(* Logix 5000 project; controller test4 1769-L16ER-BB1B rev 36.11; software revision 36.00 *)

TASK MainTask (continuous, watchdog 500 ms) : MainProgram

MODULES
   Local : 1769-L16ER-BB1B (PointIO 0, rev 36.11)
      Discrete_IO : Embedded (PointIO 1, rev 36.11, Output RPI 20 ms)
           Local:1:I.Data.1   // Button 2
           Local:1:I.Data.2   // Button 3
           Local:1:I.Data.3   // Button 4
           Local:1:I.Data.4   // Switch 1
           Local:1:O.Data.0   // Light 1
           Local:1:O.Data.1   // Light 2
END_MODULES

PROGRAM MainProgram   (* main routine MainRoutine *)
VAR
   Green_Button : ALIAS FOR Local:1:I.Data.0;
   GreenButton : ALIAS FOR Local:1:I.Data.0;
   Timer1 : TIMER := (PRE := 4000, ACC := 1);
END_VAR

ROUTINE FBD1   (* function block diagram *)
   SHEET 1
END_ROUTINE

ROUTINE MainRoutine   (* ladder *)
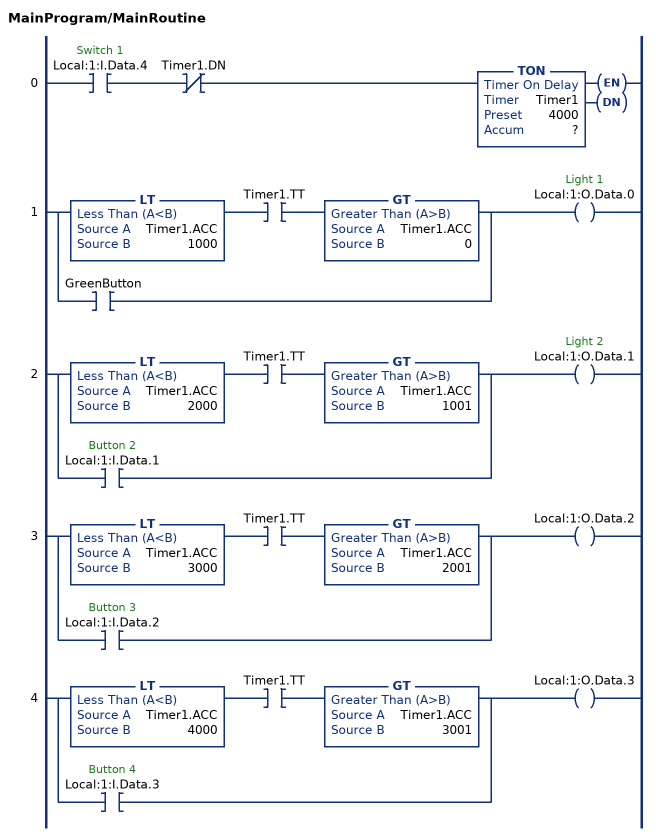
   0: XIC(Local:1:I.Data.4)XIO(Timer1.DN)TON(Timer1,?,?);
   1: [LT(Timer1.ACC,1000) XIC(Timer1.TT) GT(Timer1.ACC,0) ,XIC(GreenButton) ]OTE(Local:1:O.Data.0);
   2: [LT(Timer1.ACC,2000) XIC(Timer1.TT) GT(Timer1.ACC,1001) ,XIC(Local:1:I.Data.1) ]OTE(Local:1:O.Data.1);
   3: [LT(Timer1.ACC,3000) XIC(Timer1.TT) GT(Timer1.ACC,2001) ,XIC(Local:1:I.Data.2) ]OTE(Local:1:O.Data.2);
   4: [LT(Timer1.ACC,4000) XIC(Timer1.TT) GT(Timer1.ACC,3001) ,XIC(Local:1:I.Data.3) ]OTE(Local:1:O.Data.3);
END_ROUTINE

ROUTINE ST1   (* structured text *)
   
END_ROUTINE
END_PROGRAM
